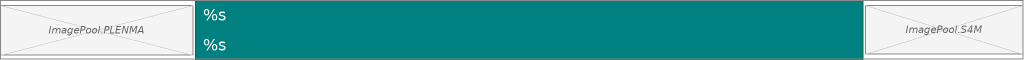
VISUALIZATION N_Header  // 1024x60
    Image (0,5 193x50), image: ImagePool.PLENMA
        OnMouseClick: VisuUserMgmt Type=Logout
    Image (865,5 158x49), image: ImagePool.S4M
    Rectangle (195,0 668x60)
    Textfield (200,0 150x30), "%s", text variable: Onlyday
    Textfield (200,30 150x30), "%s", text variable: OnlyTime
END_VISUALIZATION

(* stored: Version 1.1.0.1, ProductVersion 3.1.4024.12
   Visu N_Header: Id {39bb2ce1-8546-4b89-abbb-adbf1784d5f5} *)
